(* PLC project 未命名, 未知 未命名 1 *)
(* stored: creationDateTime 2023-06-26T21:53:33, modificationDateTime 2023-06-27T23:10:51 *)

PROGRAM program0
  VAR_INPUT
    RUN_BUTTON : BOOL;
  END_VAR
  VAR_OUTPUT
    stop_status : BOOL;
  END_VAR
  VAR_INPUT
    STOP_BUTTON : BOOL;
    BT_IN : INT;
    ET_IN : INT;
  END_VAR
  VAR_OUTPUT
    RUN_STATUS : BOOL;
  END_VAR
  VAR
    TON0 : TON;
  END_VAR

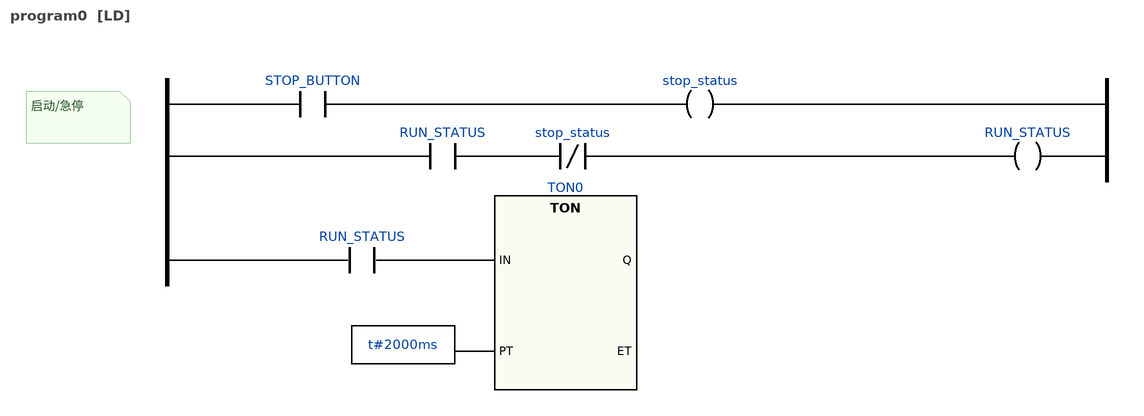
(* LD diagram, written out as Structured Text *)
(* 启动/急停 *)
stop_status := STOP_BUTTON;
RUN_STATUS := RUN_STATUS AND NOT stop_status;
TON0(IN := RUN_STATUS, PT := t#2000ms);
END_PROGRAM

CONFIGURATION Config0
  RESOURCE Res0 ON PLC
    TASK task0(INTERVAL := T#20ms, PRIORITY := 0);
    PROGRAM instance0 WITH task0 : program0;
  END_RESOURCE
END_CONFIGURATION
